FUNCTION_BLOCK SOE (* Sequence of Events *)
  (* Standard: 61499-2 *)
  (* Version 0.2, 2003-12-04, JHC, Rockwell Automation, Renamed for better indexing. *)
  (* Version 0.1, 2002-11-05, JHC, Rockwell Automation, Corrected missing ST element in Algorithm REQ. *)
  (* Version 0.0, 2000-05-30, JHC, Rockwell Automation *)
  (* Compiler header: package fb.rt.student; *)
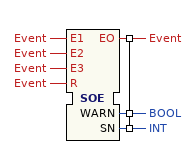
  EVENT_INPUT
    E1; (* Initialization Request *)
    E2; (* Normal Execution Request *)
    E3;
    R; (* RESET *)
  END_EVENT
  EVENT_OUTPUT
    EO WITH WARN, SN; (* State Change Notification *)
  END_EVENT
  VAR_OUTPUT
    WARN : BOOL; (* WARNING - Sequence E1,E2,E3 Detected! *)
    SN : INT; (* State Number = {0,1,2,3} *)
  END_VAR
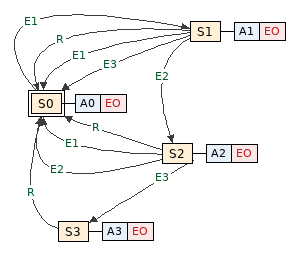
  EC_STATES
    S0 : A0 -> EO; (* Initial State *)
    S1 : A1 -> EO; (* E1 detected *)
    S2 : A2 -> EO; (* E1, E2 detected *)
    S3 : A3 -> EO; (* WARNING - E1,E2,E3 detected *)
  END_STATES
  EC_TRANSITIONS
    S0 TO S1 := E1;
    S1 TO S0 := R;
    S3 TO S0 := R;
    S2 TO S0 := R;
    S1 TO S2 := E2;
    S2 TO S3 := E3;
    S1 TO S0 := E1;
    S1 TO S0 := E3;
    S2 TO S0 := E1;
    S2 TO S0 := E2;
  END_TRANSITIONS
  ALGORITHM A0 IN ST: (* Algorithm for S0 *)
SN := 0;
WARN := FALSE;
  END_ALGORITHM
  ALGORITHM A1 IN ST: (* Algorithm for S1 *)
SN := 1;
  END_ALGORITHM
  ALGORITHM A2 IN ST: (* Algorithm for S2 *)
SN := 2;
  END_ALGORITHM
  ALGORITHM A3 IN ST: (* WARNING algorithm for S3 *)
SN := 3;
WARN := TRUE;
  END_ALGORITHM
END_FUNCTION_BLOCK
